// TwinCAT 3 PLC project Main
// ProgramVersion: 3.1.4023.0
// libraries:
//   mobject-packml, * (mobject.io)
//   Tc2_Standard, * (Beckhoff Automation GmbH)
//   Tc2_System, * (Beckhoff Automation GmbH)
//   Tc3_Module, * (Beckhoff Automation GmbH)
//   TcUnit, * (www.tcunit.org)
// project tree:
//   / PlcTask.TcTTO
//   POUs/ MAIN.TcPOU
//   POUs/SimplePackMLModeExample/ SimpleMachine.TcPOU
//   Tests/ TEST_PRG.TcPOU
// real-time tasks:
//   TASK PlcTask: cycle T#10ms, priority 20, ADS port 350

CONFIGURATION Main
    RESOURCE PLC ON TwinCAT3
        TASK PlcTask(INTERVAL := T#10ms, PRIORITY := 20);
        PROGRAM MAIN WITH PlcTask : MAIN;
    END_RESOURCE
END_CONFIGURATION

// ---- POUs/MAIN.TcPOU
PROGRAM MAIN
VAR
	
	start : BOOL;
	stop : BOOL;
	abort : BOOL;
	reset : BOOL;
	clear : BOOL;
	hold : BOOL;
	unhold : BOOL;
	suspend : BOOL;
	unsuspend : BOOL;
	
	currentState : PackML_State;

	simpleMachine : SimpleMachine;
	
END_VAR

IF start THEN
	start := FALSE;
	simpleMachine.Start();
END_IF

IF stop THEN
	stop := FALSE;
	simpleMachine.Stop();
END_IF

IF reset THEN
	reset := FALSE;
	simpleMachine.Reset();
END_IF

IF abort THEN
	abort := FALSE;
	simpleMachine.Abort();
END_IF

IF clear THEN
	clear := FALSE;
	simpleMachine.Clear();
END_IF

IF hold THEN
	hold := FALSE;
	simpleMachine.Hold();
END_IF

IF unhold THEN
	unhold := FALSE;
	simpleMachine.Unhold();
END_IF

IF suspend THEN
	suspend := FALSE;
	simpleMachine.Suspend();
END_IF

IF unsuspend THEN
	unsuspend := FALSE;
	simpleMachine.Unsuspend();
END_IF

currentState := simpleMachine.CurrentState;

// remember you can also couple this with mobject-core to make this a self calling cyclic instance.  
// Checkout the documents to find out how.
simpleMachine.CyclicCall();

END_PROGRAM

// ---- POUs/SimplePackMLModeExample/SimpleMachine.TcPOU
FUNCTION_BLOCK SimpleMachine EXTENDS PackML_Mode
VAR
	executeTimer : ton;
END_VAR

METHOD PROTECTED Execute
VAR_INPUT
	Commands : I_PackML_ExecuteCommands;
END_VAR
// in the execute state we will wait for the timer to elapse before continuing to the next state

executeTimer(in:=TRUE,pt:=T#2S);

IF executeTimer.Q THEN
	Commands.StateComplete();
END_IF
END_METHOD

METHOD PROTECTED Starting
VAR_INPUT
	Commands : I_PackML_StartingCommands;
END_VAR
// in the starting transition state we will reset the timer and then trigger the next state

executeTimer(in:=FALSE);
Commands.StateComplete();
END_METHOD

END_FUNCTION_BLOCK

// ---- Tests/TEST_PRG.TcPOU
PROGRAM TEST_PRG
VAR
END_VAR

TcUnit.RUN();

END_PROGRAM
